FUNCTION Convert_USINT_TO_BOOL : Hresult
VAR_INPUT
	in : USINT;
	out : REFERENCE TO BOOL;
END_VAR
VAR
	converted : BOOL;
END_VAR
VAR CONSTANT
	INCOMPATIBLE : HRESULT := 16#9811070E;
END_VAR

converted := USINT_TO_BOOL(in);

IF (BOOL_TO_USINT(converted) <> in) THEN
	Convert_USINT_TO_BOOL := INCOMPATIBLE;
	RETURN;
END_IF

out := converted;

END_FUNCTION

(* stored: Version 1.1.0.1, ProductVersion 3.1.4024.12
   POU Convert_USINT_TO_BOOL: Id {5ec0b8a0-daac-4744-bfc8-629e3b62234d}, SpecialFunc None *)
